% RSLogix 500 project PROJECT7.RSS, saved by version 8.30.00.16 %
PROJECT "PROJECT7"    % processor: Bul.1763 MicroLogix 1100 Series B %

PROGRAM FILES
  LAD 2 "MAIN"  5 rungs
  LAD 3 "I/O"  5 rungs
  LAD 4 "CONTROL"  3 rungs
  LAD 5 "CALIBRATE"  8 rungs

DATA FILES
  O0 OUTPUT  5 elements
  I1 INPUT  6 elements
  S2 STATUS  66 elements
  B3 BINARY  1 elements
  T4 TIMER  4 elements
  C5 COUNTER  2 elements
  R6 CONTROL  1 elements
  N7 INTEGER  8 elements
  F8 FLOAT  8 elements

LADDER 2 "MAIN"
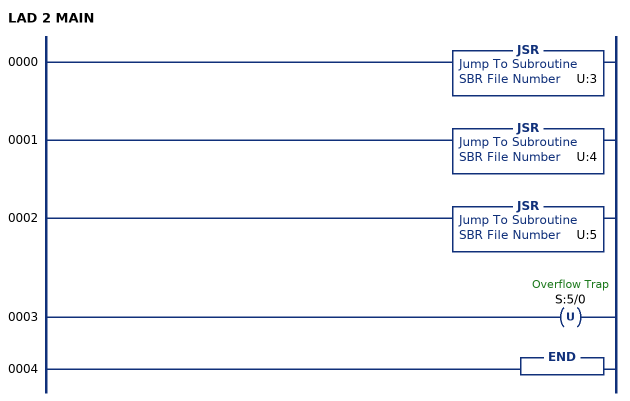
% Rung: 0 %
SOR JSR U:3 EOR
% Rung: 1 %
SOR JSR U:4 EOR
% Rung: 2 %
SOR JSR U:5 EOR
% Rung: 3 %
SOR OTU S:5/0 EOR
%   S:5/0  "Overflow Trap" %
% Rung: 4 %
SOR END EOR

LADDER 3 "I/O"
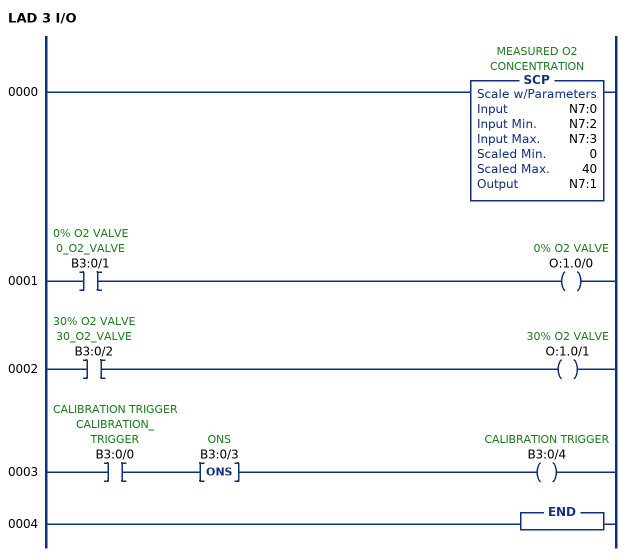
% Rung: 0 %
SOR SCP N7:0 N7:2 N7:3 0 40 N7:1 EOR
%   N7:0  "O2 INPUT" %
%   N7:2  "INPUT MIN" %
%   N7:3  "INPUT MAX" %
%   N7:1  "MEASURED O2 CONCENTRATION" %
% Rung: 1 %
SOR XIC B3:0/1 OTE O:1.0/0 EOR
%   B3:0/1  0_O2_VALVE  "0% O2 VALVE" %
%   O:1.0/0  "0% O2 VALVE" %
% Rung: 2 %
SOR XIC B3:0/2 OTE O:1.0/1 EOR
%   B3:0/2  30_O2_VALVE  "30% O2 VALVE" %
%   O:1.0/1  "30% O2 VALVE" %
% Rung: 3 %
SOR XIC B3:0/0 ONS B3:0/3 OTE B3:0/4 EOR
%   B3:0/0  CALIBRATION_TRIGGER  "CALIBRATION TRIGGER" %
%   B3:0/3  "ONS" %
%   B3:0/4  "CALIBRATION TRIGGER" %
% Rung: 4 %
SOR END EOR

LADDER 4 "CONTROL"
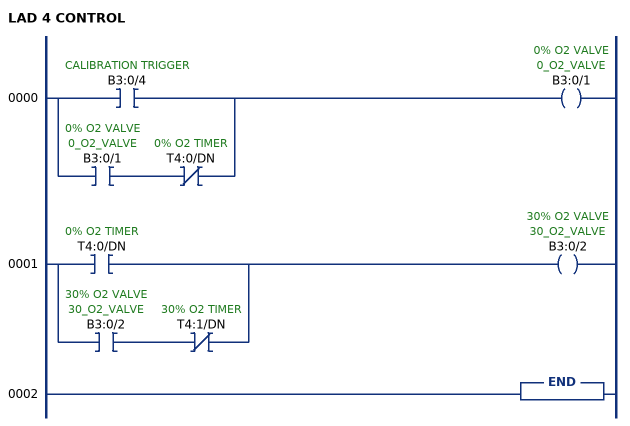
% Rung: 0 %
SOR BST XIC B3:0/4 NXB XIC B3:0/1 XIO T4:0/DN BND OTE B3:0/1 EOR
%   B3:0/4  "CALIBRATION TRIGGER" %
%   B3:0/1  0_O2_VALVE  "0% O2 VALVE" %
%   T4:0  "0% O2 TIMER" %
% Rung: 1 %
SOR BST XIC T4:0/DN NXB XIC B3:0/2 XIO T4:1/DN BND OTE B3:0/2 EOR
%   T4:0  "0% O2 TIMER" %
%   B3:0/2  30_O2_VALVE  "30% O2 VALVE" %
%   T4:1  "30% O2 TIMER" %
% Rung: 2 %
SOR END EOR

LADDER 5 "CALIBRATE"
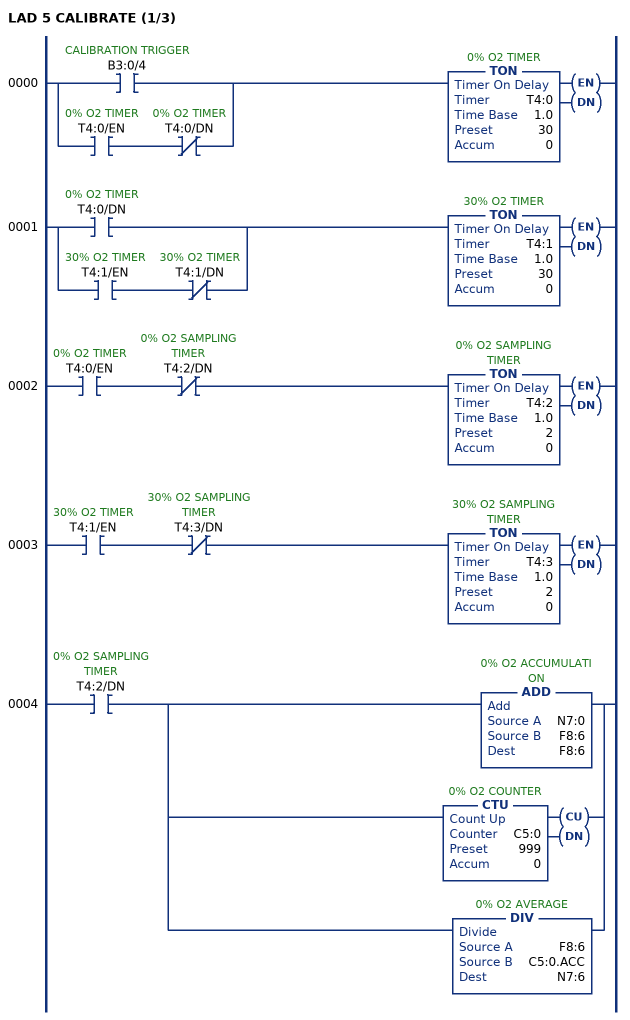
% Rung: 0 %
SOR BST XIC B3:0/4 NXB XIC T4:0/EN XIO T4:0/DN BND TON T4:0 1.0 30 0 EOR
%   B3:0/4  "CALIBRATION TRIGGER" %
%   T4:0  "0% O2 TIMER" %
% Rung: 1 %
SOR BST XIC T4:0/DN NXB XIC T4:1/EN XIO T4:1/DN BND TON T4:1 1.0 30 0 EOR
%   T4:0  "0% O2 TIMER" %
%   T4:1  "30% O2 TIMER" %
% Rung: 2 %
SOR XIC T4:0/EN XIO T4:2/DN TON T4:2 1.0 2 0 EOR
%   T4:0  "0% O2 TIMER" %
%   T4:2  "0% O2 SAMPLING TIMER" %
% Rung: 3 %
SOR XIC T4:1/EN XIO T4:3/DN TON T4:3 1.0 2 0 EOR
%   T4:1  "30% O2 TIMER" %
%   T4:3  "30% O2 SAMPLING TIMER" %
% Rung: 4 %
SOR XIC T4:2/DN BST ADD N7:0 F8:6 F8:6 NXB CTU C5:0 999 0 NXB DIV F8:6 C5:0.ACC N7:6 BND EOR
%   T4:2  "0% O2 SAMPLING TIMER" %
%   N7:0  "O2 INPUT" %
%   F8:6  "0% O2 ACCUMULATION" %
%   C5:0  "0% O2 COUNTER" %
%   N7:6  "0% O2 AVERAGE" %

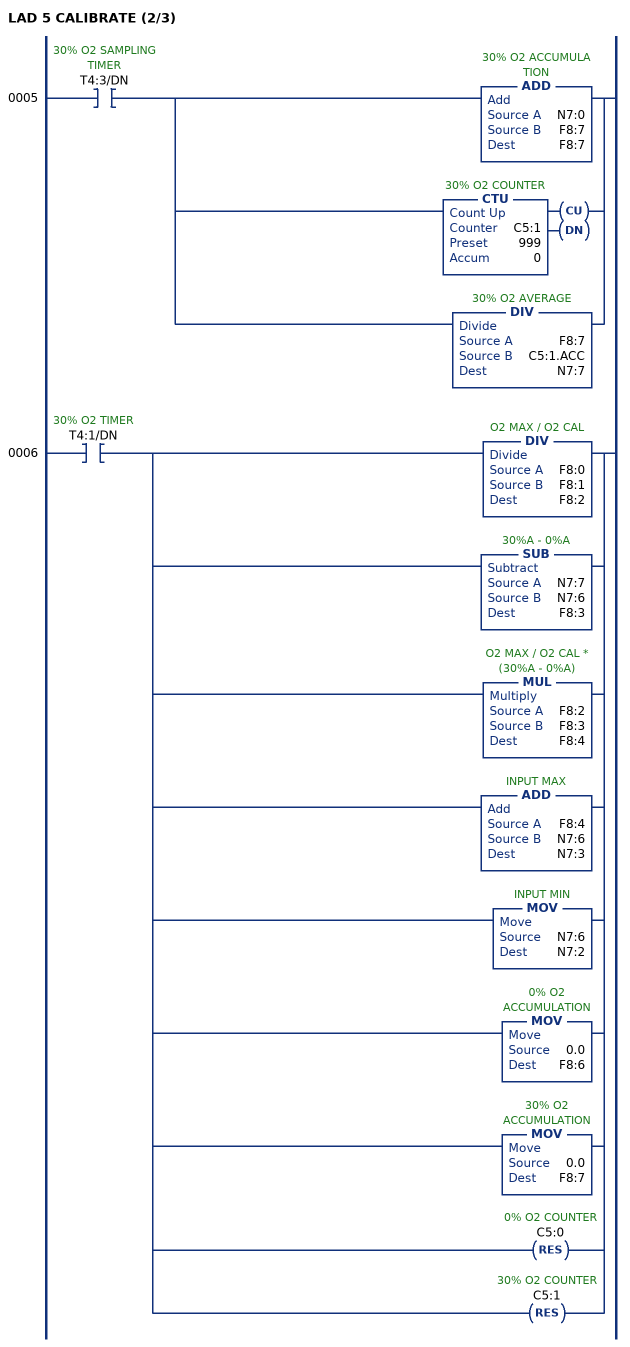
% Rung: 5 %
SOR XIC T4:3/DN BST ADD N7:0 F8:7 F8:7 NXB CTU C5:1 999 0 NXB DIV F8:7 C5:1.ACC N7:7 BND EOR
%   T4:3  "30% O2 SAMPLING TIMER" %
%   N7:0  "O2 INPUT" %
%   F8:7  "30% O2 ACCUMULATION" %
%   C5:1  "30% O2 COUNTER" %
%   N7:7  "30% O2 AVERAGE" %
% Rung: 6 %
SOR XIC T4:1/DN BST DIV F8:0 F8:1 F8:2 NXB SUB N7:7 N7:6 F8:3 NXB MUL F8:2 F8:3 F8:4 NXB ADD F8:4 N7:6 N7:3 NXB MOV N7:6 N7:2 NXB MOV 0.0 F8:6 NXB MOV 0.0 F8:7 NXB RES C5:0 NXB RES C5:1 BND EOR
%   T4:1  "30% O2 TIMER" %
%   F8:0  "O2 MAX CONCENTRATION" %
%   F8:1  "O2 CALIBRATION CONCENTRATION" %
%   F8:2  "O2 MAX / O2 CAL" %
%   N7:7  "30% O2 AVERAGE" %
%   N7:6  "0% O2 AVERAGE" %
%   F8:3  "30%A - 0%A" %
%   F8:4  "O2 MAX / O2 CAL * (30%A - 0%A)" %
%   N7:3  "INPUT MAX" %
%   N7:2  "INPUT MIN" %
%   F8:6  "0% O2 ACCUMULATION" %
%   F8:7  "30% O2 ACCUMULATION" %
%   C5:0  "0% O2 COUNTER" %
%   C5:1  "30% O2 COUNTER" %

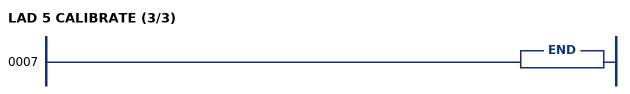
% Rung: 7 %
SOR END EOR

OTHER DOCUMENTED ADDRESSES
  B3:0/5  "CALIBRATION RUNNING"
  B3:0/6  "CALIBRATION INTERRUPT"
  F8:5  "INPUT MAX"
  N7:4  "0% O2 ACCUMULATION"
  N7:5  "30% O2 ACCUMULATION"
  O:0.0/0  "0% VALVE"

DATA TABLE (non-zero values as saved)
DATA T4
% .PRE .ACC %
% T4:0 % 30 0
% T4:1 % 30 0
% T4:2 % 2 0
% T4:3 % 2 0
DATA C5
% .PRE .ACC %
% C5:0 % 999 0
% C5:1 % 999 0
DATA N7
% N7:0 % 0 0 0 16383 0 0 0 0
DATA F8
% F8:0 % 40 30 0 0 0
